// TwinCAT 3 PLC project Main
// ProgramVersion: 3.1.4024.0
// libraries:
//   Tc2_EtherCAT, * (Beckhoff Automation GmbH)
//   Tc2_IoFunctions, * (Beckhoff Automation GmbH)
//   Tc2_Math, * (Beckhoff Automation GmbH)
//   Tc2_MC2, * (Beckhoff Automation GmbH)
//   Tc2_NC, * (Beckhoff Automation GmbH)
//   Tc2_Standard, * (Beckhoff Automation GmbH)
//   Tc2_System, * (Beckhoff Automation GmbH)
//   Tc2_Utilities, * (Beckhoff Automation GmbH)
//   Tc3_EventLogger, * (Beckhoff Automation GmbH)
//   Tc3_McCollisionAvoidance, * (Beckhoff Automation GmbH)
//   Tc3_McCoordinatedMotion, * (Beckhoff Automation GmbH)
//   Tc3_Module, * (Beckhoff Automation GmbH)
//   Tc3_XTS_Utility, * (Beckhoff Automation GmbH)
//   VisuDialogs, * (System)
//   VisuSymbols,3.5.10.0,System
// project tree:
//   DUTs/ MainCommands_typ.TcDUT (not stored), MainStateMachine_enum.TcDUT (not stored), MainState_enum.TcDUT (not stored), MediatorGroupStatus.TcDUT (not stored), MoverCommandType_enum.TcDUT (not stored), MotionParameters_typ.TcDUT (not stored), MoverState_enum.TcDUT (not stored), PositionTriggerStats_typ.TcDUT (not stored), StationStats_typ.TcDUT (not stored), TrackCyclicState.TcDUT (not stored), TrackInfo.TcDUT (not stored), TrackState.TcDUT (not stored), UserStationsMonitor.TcDUT
//   / GlobalTextList.TcGTLO (not stored), PlcTask.TcTTO (not stored), Visualization Manager.TcVMO (not stored)
//   GVLs/ GVL.TcGVL, SAFETY.TcGVL
//   ITFs/ iMoverList.TcIO (not stored), iMover.TcIO (not stored), iTrack.TcIO (not stored)
//   POUs/ MAIN.TcPOU
//   POUs/XTS/Administrative/ ErrorMover.TcPOU (not stored), Mediator.TcPOU (not stored), Objective.TcPOU (not stored)
//   POUs/XTS/ Mover.TcPOU (not stored), MoverList.TcPOU (not stored), PositionTrigger.TcPOU (not stored), Station.TcPOU (not stored), Track.TcPOU (not stored), Zone.TcPOU (not stored)
//   VISUs/ Controls.TcVIS (not stored), DiagnosticVisu.TcVIS (not stored)

// ---- DUTs/UserStationsMonitor.TcDUT
TYPE UserStationsMonitor :
STRUCT
	
bmoverAtStation		: ARRAY[0..GVL.NUM_STATIONS] OF BOOL;
nmoverAtStation		: ARRAY[0..GVL.NUM_STATIONS] OF UDINT;


END_STRUCT
END_TYPE

// ---- GVLs/GVL.TcGVL
{attribute 'qualified_only'}
VAR_GLOBAL CONSTANT

	TRACK_LENGTH 			: LREAL := 7000; // This should be set to the exact length [mm] of the track system
		
	NUM_MOVERS   			: USINT := 20;   // This should be set to the exact number of movers on the system
	
	// The following should be set to a value **equal to or greater than** the number of objectives needed
	NUM_MOVERLISTS			: USINT := 10;	// Mover Lists
	NUM_POSITIONTRIGGERS	: USINT := 10;	// Position Triggers
	NUM_STATIONS			: USINT := 10;	// Stations
	NUM_ZONES				: USINT := 10;	// Zones
	
	NUM_TRACKS				: USINT	:= 1;	// Tracks (Typically 1)

	PART_ARRAY_SIZE			: UDINT := 100;
	AUTO_POPULATE_STATIONS  : BOOL := TRUE; // use the Station[x] array to label stations on the visualization. Turn off if manually entering stations in the configurator.
	
	// statistics weighted average
	ALPHA_EMA				: LREAL := 0.1;

END_VAR
VAR_GLOBAL
	newCallTime: LREAL;
END_VAR

// ---- GVLs/SAFETY.TcGVL
{attribute 'qualified_only'}
VAR_GLOBAL
	

err_ack		AT %Q*	:	BOOL;
run			AT %Q*	:	BOOL;

bEstopSet	AT %I*	:	BOOL;

END_VAR

// ---- POUs/MAIN.TcPOU
PROGRAM MAIN
VAR	

	// ========= System Control / FSM Variables =========
	
	MainCommands 		: MainCommands_typ; 		// command struct for cycling thru the state machine
	MainState    		: MainStateMachine_enum;   	// enumeration for the Main state machine
	System				: Mediator;					// System-level control object

	// ========= Linked NC Variables & References =========
	
	Mover    			: ARRAY[1..GVL.NUM_MOVERS] OF Mover; 	// instantiation of Mover objects. Matches the number of movers on the system
	
	// ========= Objectives & Parameters =========

	ParameterSet		: MotionParameters_typ;
	
	MoverList			: ARRAY[0..GVL.NUM_MOVERLISTS-1] OF MoverList;
	PositionTrigger		: ARRAY[0..GVL.NUM_POSITIONTRIGGERS-1] OF PositionTrigger;
	Station				: ARRAY[0..GVL.NUM_STATIONS-1] OF Station;
	Track				: ARRAY[0..GVL.NUM_TRACKS] OF Track;
	Zone				: ARRAY[0..GVL.NUM_ZONES-1] OF Zone;
	
    // ========= Helper, State, & Index Variables =========
	
    i                	: UINT; 	// index variable; gets reused in various FOR loops
    n                	: UINT; 	// secondary index variable, for enabling movers
	
	// ========= Example Application Variables =========

    lowVelocity    		: LREAL := 200;  	// mm/s
    mediumVelocity 		: LREAL := 800;  	// mm/s
    highVelocity   		: LREAL := 1200; 	// mm/s
	
	userStationsMonitor	: UserStationsMonitor;
	
	trigUP1				: R_TRIG;
	trigDOWN1			: F_TRIG;
	
	loadTray_Busy			: 	BOOL;
	firstRun				:	BOOL;
	loadTray_Complete		:	BOOL;
	loadArea1_Busy			:	BOOL;
	loadArea1_Complete		: 	BOOL;
	loadArea2_Busy			: 	BOOL;
	loadArea2_Complete		: 	BOOL;
	loadArea3_Busy			: 	BOOL;
	loadArea3_Complete		:   BOOL;
	loadArea4_Busy			: 	BOOL;
	loadArea4_Complete		: 	BOOL;
	unloadTray_Busy			:	BOOL;
	unloadTray_Complete		:	BOOL;
	zone0Stop				:	BOOL;
	bOneShotConstantVel		:	BOOL;
	iConstantSpeedVel		:	INT;
	bOneShotMove			:	BOOL;
	iStationLoop			:	INT;
END_VAR


CASE MainState OF
	MainStateMachine_enum.MS_DISABLED: // ------------------------------------------
	
		// XTS is idle. Motive power is disabled.	
		IF MainCommands.Enable THEN
			MainCommands.Disable			:= FALSE;
			MainCommands.Stop				:= FALSE;
			MainState						:= MainStateMachine_enum.MS_INITIALIZING;
		END_IF

	MainStateMachine_enum.MS_INITIALIZING: // --------------------------------------
	
		Registering();			// Add all objectives & movers to the system-level Mediator object
		Initializing();			// Set basic application parameters for the objects
			
		System.CompleteMoverList.EnableAll();
		System.CompleteMoverList.ActivateAllTrack( Track[1] );
		
		IF System.CompleteMoverList.IsAllTrackReady AND System.CompleteMoverList.IsAllMoversReady THEN
			MainState	:= MainStateMachine_enum.MS_ENABLED;
		END_IF
		
		IF MainCommands.Disable THEN
			MainCommands.Enable	:= FALSE;
			System.CompleteMoverList.DisableAll();
			MainState			:= MainStateMachine_enum.MS_DISABLING;
		END_IF
	
	MainStateMachine_enum.MS_ENABLED:	// -------------------------------------------
	
		// Recovery logic
		IF MainCommands.Start THEN
			System.CompleteMoverList.SetAllVelocity(mediumVelocity).MoveAllToStation( Station[0] );
			System.ResetStatistics();
			MainState			:= MainStateMachine_enum.MS_RUN;
		ELSIF MainCommands.Disable THEN
			MainCommands.Enable	:= FALSE;
			System.CompleteMoverList.HaltAll();
			MainState			:= MainStateMachine_enum.MS_STOPPING;
			
		END_IF
	
	MainStateMachine_enum.MS_RUN: // -----------------------------------------------
	
		StationLogic();
        IF System.GroupError THEN
			// stop on group error user must go through disable/enable to recover
			MainCommands.Start	:= FALSE;
			MainState 			:= MainStateMachine_enum.MS_STOPPING;
		ELSIF MainCommands.Stop THEN
            MainCommands.Start 	:= FALSE;
			System.CompleteMoverList.HaltAll();
            MainState         	:= MainStateMachine_enum.MS_STOPPING;
        ELSIF MainCommands.Disable THEN
            MainCommands.Enable := FALSE;
			System.CompleteMoverList.HaltAll();
            MainState           := MainStateMachine_enum.MS_STOPPING;
        END_IF
		
	MainStateMachine_enum.MS_STOPPING:
	
		IF System.CompleteMoverList.IsAllMoversHalted THEN
			MainState			:= MainStateMachine_enum.MS_STOPPED;
		END_IF
		
	MainStateMachine_enum.MS_STOPPED: // -------------------------------------------
	
	    IF MainCommands.Disable THEN
            MainCommands.Enable 	:= FALSE;
			MainCommands.Start		:= FALSE;
			MainCommands.Stop		:= FALSE;
			System.CompleteMoverList.DisableAll();
            MainState           	:= MainStateMachine_enum.MS_DISABLING;
        ELSIF MainCommands.Start THEN
            MainCommands.Stop 		:= FALSE;
            MainState         		:= MainStateMachine_enum.MS_ENABLED;
        END_IF
		
	MainStateMachine_enum.MS_DISABLING: // -------------------------------------------
	
		IF System.CompleteMoverList.IsAllMoversDisabled THEN
			MainState			:= MainStateMachine_enum.MS_DISABLED;
		END_IF
		
	MainStateMachine_enum.MS_ERROR: // ---------------------------------------------
	MainStateMachine_enum.MS_DEBUG: // ---------------------------------------------	
	

END_CASE

System.Cyclic();

ACTION Initializing:


	// Initialize station positions
	Station[0].Position 		:= 1275;					//Load Tray Beginning
	Station[1].Position 		:= 2820;					//Load Parts Section 1
	Station[2].Position 		:= 3446;					//Load Parts Section 2
	Station[3].Position 		:= 4060;					//Load Parts Section 3
	Station[4].Position 		:= 4686;					//Load Parts Section 4
	Station[5].Position 		:= 5500;					//Unload Tray End

	PositionTrigger[0].Position := 1300;
	PositionTrigger[1].Position := 5500;
	PositionTrigger[2].Position := 3500;

	Zone[0].StartPosition		:= 5600;
	Zone[0].EndPosition   		:= 1275;

	Zone[1].StartPosition 		:= 1275;
	Zone[1].EndPosition   		:= 5600;

	// testing zone used for recovery
	Zone[2].StartPosition 		:= 1225;
	Zone[2].EndPosition   		:= 1325;

	Zone[3].StartPosition		:= 2750;
	Zone[3].EndPosition   		:= 3750;
	
	System.CompleteMoverList.SetAllVelocity( 1E3 );
	System.CompleteMoverList.SetAllAcceleration( 1E4 );
	System.CompleteMoverList.SetAllDeceleration( 1E4 );
	System.CompleteMoverList.SetAllJerk( 5E5 );
	System.CompleteMoverList.SetAllGap( 200 );
	System.CompleteMoverList.SetAllDirection( mcDirectionPositive );
END_ACTION

ACTION LightCurtainZone0Stop:


	trigUP1(CLK := zone0Stop);
	trigDOWN1(CLK := zone0Stop);
		
	IF trigUP1.Q THEN
		zone[0].CurrentMoverList.SetAllVelocity(0.1);
	END_IF
	
	IF trigDOWN1.Q THEN
		zone[0].CurrentMoverList.SetAllVelocity(lowVelocity);
	END_IF
END_ACTION

ACTION Registering:
	

		// Add all Movers to the Mediator
		FOR i := 1 TO GVL.NUM_MOVERS DO
			System.AddMover( Mover[i] );
		END_FOR
	
		// Add all Mover Lists to the Mediator
		FOR i := 0 TO GVL.NUM_MOVERLISTS - 1 DO
			System.AddMoverList( MoverList[i] );
		END_FOR
		
		// Add all PositionTriggers to the Mediator
		FOR i := 0 TO GVL.NUM_POSITIONTRIGGERS - 1 DO
			System.AddPositionTrigger( PositionTrigger[i] );
		END_FOR
		
		// Add all Stations to the Mediator
		FOR i := 0 TO GVL.NUM_STATIONS - 1 DO
			System.AddStation( Station[i] );
		END_FOR
		
		// Add all Tracks to the Mediator
		// note track zero is a special case, so the loop is one larger than the rest of the initalization loops
		FOR i := 0 TO GVL.NUM_TRACKS DO
			Track[i].Id := UINT_TO_INT(i);
			System.AddTrack( Track[i] );
		END_FOR
		
		// Add all Zones to the Mediator
		FOR i := 0 TO GVL.NUM_ZONES - 1 DO
			System.AddZone( Zone[i] );
		END_FOR
END_ACTION

ACTION SpeedControl:
//Changes the speeds of movers as they enter/leave loading area

       // Position Trigger 0 Logic
        IF PositionTrigger[0].MoverPassedPosition THEN
            PositionTrigger[0].CurrentMover.SetVelocity(mediumVelocity);
            PositionTrigger[0].MuteCurrent();
        END_IF
	
		        // Position Trigger 1 Logic
        IF PositionTrigger[1].MoverPassedPosition THEN
            PositionTrigger[1].CurrentMover.SetVelocity(lowVelocity);
            PositionTrigger[1].MuteCurrent();
        END_IF
END_ACTION

ACTION StationLogic:
		(*Mover routing logic should be written here to define the system's operating behavior.
		Station implementations, Position Trigger logic, etc. In general, you can remove the example code
		here down to the short line break that looks like this: // ============= *)

	
		//-----------------------------------------------------------LOADING TRAYS--------------------------------------------------

	IF Station[0].MoverInPosition THEN
    	loadTray_Busy := TRUE;
		firstRun := TRUE;
    	IF loadTray_Complete THEN
        	Station[0].CurrentMover.MoveToStation( Station[1] );
			loadTray_Complete := FALSE;  
			loadTray_Busy := FALSE;
    	END_IF
	END_IF
	
	
	//-----------------------------------------------------------LOADING Parts 1--------------------------------------------------
	IF Station[1].MoverInPosition AND firstRun THEN
    	loadArea1_Busy := TRUE;
    	IF loadArea1_Complete THEN
        	Station[1].CurrentMover.MoveToStation( Station[2] );
			loadArea1_Complete := FALSE;
			loadArea1_Busy := FALSE;
    	END_IF
	END_IF
	
	//-----------------------------------------------------------LOADING Parts 2--------------------------------------------------
	IF Station[2].MoverInPosition AND firstRun  THEN
    	loadArea2_Busy := TRUE;
    	IF loadArea2_Complete THEN
			//station3MoverID := Station[3].CurrentMover;
        	Station[2].CurrentMover.MoveToStation( Station[3] );
			loadArea2_Complete := FALSE;
			loadArea2_Busy := FALSE;
    	END_IF
	END_IF
	
	//-----------------------------------------------------------LOADING Parts 3--------------------------------------------------
	IF Station[3].MoverInPosition AND firstRun THEN
    	loadArea3_Busy := TRUE;
    	IF loadArea3_Complete THEN
			//station4MoverID := Station[4].CurrentMover;
        	Station[3].CurrentMover.MoveToStation( Station[4] );
			loadArea3_Complete := FALSE;
			loadArea3_Busy := FALSE;
    	END_IF
	END_IF
	
	//-----------------------------------------------------------LOADING Parts 4--------------------------------------------------
	IF Station[4].MoverInPosition AND firstRun THEN
    	loadArea4_Busy := TRUE;
    	IF loadArea4_Complete THEN
			//station5MoverID := Station[5].CurrentMover;
        	Station[4].CurrentMover.MoveToStation( Station[5] );
			loadArea4_Complete := FALSE;
			loadArea4_Busy := FALSE;
    	END_IF
	END_IF
	
	
	//-----------------------------------------------------------UNLOADING TRAY--------------------------------------------------
	IF Station[5].MoverInPosition AND firstRun THEN
    	unloadTray_Busy := TRUE;
    	IF unloadTray_Complete THEN
			//station6MoverID := Station[6].CurrentMover;
        	Station[5].CurrentMover.MoveToStation( Station[0] );
			unloadTray_Complete := FALSE;
			unloadTray_Busy := FALSE;
    	END_IF
	END_IF
	
	
	LightCurtainZone0Stop();
	
    SpeedControl();
	
	//Move at constant velocity
	IF bOneShotConstantVel THEN
		System.CompleteMoverList.MoveAllVelocity(iConstantSpeedVel);
		bOneShotConstantVel := FALSE;
	END_IF
	
	//	
	IF bOneShotMove THEN
		Mover[5].MoveToPosition( 2000 );
		bOneShotMove := FALSE;
	END_IF
		
		
		(*
	
        // Station 0 Logic
        IF Station[0].MoverInPosition THEN
            StationTimer[0](IN := TRUE, PT := T#1000MS);
            IF StationTimer[0].Q THEN
                Station[0].CurrentMover.SetVelocity(mediumVelocity);
                Station[0].CurrentMover.MoveToStation(Station[1]);
            END_IF
        ELSE
            StationTimer[0](IN := FALSE);
        END_IF
		
        // Station 1 Logic		
        IF Station[1].MoverInPosition THEN
            StationTimer[1](IN := TRUE, PT := T#250MS);
            IF StationTimer[1].Q THEN
                Station[1].CurrentMover.SetVelocity(mediumVelocity);
                Station[1].CurrentMover.MoveToStation(Station[nextStation]);
                nextStation := nextStation - 1;
                IF nextStation = 1 THEN
                    nextStation := 4;
                END_IF
            END_IF
        ELSE
            StationTimer[1](IN := FALSE);
        END_IF
		
		// Group of Stations 2, 3, and 4 Logic
        IF Station[2].MoverInPosition AND Station[3].MoverInPosition AND Station[4].MoverInPosition THEN
            StationTimer[2](IN := TRUE, PT := T#750MS);
            IF StationTimer[2].Q THEN
				StationTimer[2](IN := FALSE);

                Station[2].CurrentMover.MoveVelocity(500);
                Station[3].CurrentMover.MoveVelocity(500);
                Station[4].CurrentMover.MoveVelocity(500);
            END_IF
        END_IF
		
        // Position Trigger 0 Logic
        IF PositionTrigger[0].MoverPassedPosition THEN
            PositionTrigger[0].CurrentMover.SetVelocity(lowVelocity);
            PositionTrigger[0].MuteCurrent();
        END_IF
		
        // Position Trigger 1 Logic
        IF PositionTrigger[1].MoverPassedPosition THEN
			PositionTrigger[1].CurrentMover.SetAcceleration(5E2);
            PositionTrigger[1].CurrentMover.SetVelocity(highVelocity);
            PositionTrigger[1].MuteCurrent();
        END_IF

		// Position Trigger 2 Logic
        IF PositionTrigger[2].MoverPassedPosition THEN
			PositionTrigger[2].CurrentMover.SetAcceleration(1E4);
            PositionTrigger[2].CurrentMover.SetVelocity(lowVelocity);
            PositionTrigger[2].CurrentMover.MoveToStation(Station[0]);
            PositionTrigger[2].MuteCurrent();
        END_IF
		
		*)
END_ACTION

ACTION StationMonitoring:


//Station Monitoring *************************


FOR i := 0 TO GVL.NUM_STATIONS - 1 DO
	IF Station[i].MoverInPosition THEN
		userStationsMonitor.bmoverAtStation[i] := TRUE;
		userStationsMonitor.nmoverAtStation[i] := Station[i].CurrentMover.AxisReference.NcToPlc.AxisId;
	ELSE
		userStationsMonitor.bmoverAtStation[i] := FALSE;
		userStationsMonitor.nmoverAtStation[i] := 0;
	END_IF
END_FOR
END_ACTION

END_PROGRAM
